// [Sample]
// Subscriber to a user specific weather station.
FUNCTION_BLOCK FB_BA_MyWeatherStationSub EXTENDS FB_BA_Subscriber
VAR_OUTPUT
	fWeatherTemperature	: REAL;
	fHumidity			: REAL;
	fBrightness			: REAL;
	
	bDisturb			: BOOL;
END_VAR
VAR
	{region 'General'}
		stData			: ST_BA_MyWeatherData;
	{endregion}
END_VAR

SUPER^();

// Update outputs of most important variables:
fWeatherTemperature := stData.fWeatherTemperature;
fHumidity := stData.fHumidity;
fBrightness := stData.fBrightness;

// Indicate:
// - A physical error that is really occured in the remote weather station
// - A reference error (E.g. broken ADS connection)
bDisturb := (stData.bDisturb) OR (Error);

METHOD FB_init : BOOL
VAR_INPUT
	bInitRetains : BOOL; // if TRUE, the retain variables are initialized (warm start / cold start)
	bInCopyCode : BOOL;  // if TRUE, the instance afterwards gets moved into the copy code (online change)
END_VAR
// [Hint]
// > Eigentlich wird an dieser Stelle das Profil definiert. Aber zur Übersicht wird es in "MAIN_SharedInterfaces" initialisiert.

// iProfile := SampleMyProfiles.MyWeatherStation;
END_METHOD

// Returns subscription-data (For storing read data).
METHOD GetData
VAR_OUTPUT
	pData			: PVOID;				// Pointer to subscribed data.
	nSize			: DINT;					// Size of subscribed data.
END_VAR
pData := ADR(stData);
nSize := SIZEOF(stData);
END_METHOD

METHOD PROTECTED OnValidateSubscription : BOOL
VAR_INPUT
	iPublisher			: I_BA_Publisher;
END_VAR
VAR
	_iSubWthSt			: I_BA_MyWeatherStation;
END_VAR
// Cast interface pointer (Used for a local subscription):
OnValidateSubscription := __QUERYINTERFACE(iPublisher, _iSubWthSt);
END_METHOD

END_FUNCTION_BLOCK

(* stored: Version 1.1.0.1, ProductVersion 3.1.4024.9
   POU FB_BA_MyWeatherStationSub: Id {17417506-e33f-4972-b839-5e8a66f2f355}, SpecialFunc None
   Folder [Protected] Events: Id {49e9a87b-26c9-44a3-9292-34b059a2047a}
   Folder Management: Id {3e63512f-3226-4cb2-af06-2db0d04fc38d}
   Method FB_init: Id {331ec02d-b0b0-4f1b-a128-6ee4179000dc}
   Method GetData: Id {09db79f0-a1cc-440f-b09b-f8092fbaa0a4}
   Method OnValidateSubscription: Id {b4a3d99f-a1de-4c68-9ca0-cad4df264726} *)
